FUNCTION_BLOCK FB_OutfeedConveyor
VAR CONSTANT
	sCycleStateTextDef: ARRAY[0..10]  OF STRING :=	
		['State 0: Wait for Start','1','2','3','4','5','6','7','8','9',
		'State 10: Error'];
	
	tCycleStateTimeouts: ARRAY[0..10] OF TIME := 
		[T#10S,T#10S,T#10S,T#10S,T#10S,T#10S,T#10S,T#10S,T#10S,T#10S,
		T#10S];

	sInitStateTextDef: ARRAY[0..10] OF STRING :=
		['State 0: Wait for Start',
		'State 1: Description Init State 1',
		'State 2: Description Init State 2',
		'State 3; Description Init State 3',
		'State 4; Description Init State 4',
		'State 5; Description Init State 5',
		'State 6; Error State'];

	tInitStateTimeouts: ARRAY[0..10] OF TIME := 
		[T#10S,T#10S,T#10S,T#10S,T#10S,T#10S,T#10S,T#10S,T#10S,T#10S
		,T#10S];
END_VAR
VAR_INPUT
	mxResetCycleState				: BOOL;
	mxResetInitState				: BOOL;
	mxForceInit						: BOOL; (*Reset Calibration Flag*)
	mxReset							: BOOL;	(*Reset Error*)
	mxEmergency						: BOOL;
	mxAutoMode						: BOOL; (* TRUE = Automode *)
	mxFirstCycle					: BOOL;

END_VAR
VAR_IN_OUT
	MachParameters					: ST_OutfeedConveyorMachPar;
	ProdParameters					: ST_OutfeedConveyorProdPar;
	SysParameters					: ST_OutfeedConveyorSysPar;
END_VAR
VAR_OUTPUT
	(*Errors*)
	Errors							: ST_OutfeedConveyorErrors;
	mxErrorInit						: BOOL;		(* Error, stop immediately. Initialisation neccesary *)
	mxErrorStopinPos				: BOOL;		(* Error, stop in position. Only reset neccesary *)

(* State vars *)
	mxCycleBusy						: BOOL;
	mxInitBusy						: BOOL;
	
(* Vars *)
	mxInitialized					: BOOL;
	
	mrActModPos						: LREAL;
END_VAR
VAR
(* State vars *)
	miCycleState					: INT :=0;
	miCycleOldstate					: INT :=0;
	mxCycleTransitionState			: BOOL := FALSE;
	sCycleStateText					: STRING;
	exCycleTimeOut					: BOOL;		(* Timeout for the whole programcycle *)
	CycleTimeout					: TON;
	CycleTimeOutUpFlank				: R_TRIG;
	mxCycleTimeoutEnable			: BOOL;
	CycleTime						: REAL;
	mxCycleHasError					: BOOL;
	miStopState						: INT;
	mxStartCycle					: BOOL;
	mxStopCycle						: BOOL;
	mxStopDirect					: BOOL;
	
	miInitState						: INT	:=0;
	miInitOldstate					: INT	:=0;
	mxInitTransitionState			: BOOL	:= FALSE;
	sInitStateText					: STRING;
	exInitTimeOut					: BOOL;		(* Timeout for the whole programcycle *)
	InitTimeout						: TON;
	InitTimeOutUpFlank				: R_TRIG;
	mxInitTimeoutEnable				: BOOL;
	InitTime						: REAL;
	mxInitHasError					: BOOL;
	mxStartInit						: BOOL;
	mxStopInit						: BOOL;
	
	(* Objects *)
	Belt							 : FB_NcAxis;

	mrSetpointPosition				: LREAL;
	mrActPosBeltSaved				: LREAL;
END_VAR

Error();
Cycle();
Init();
Objects();

mrActModPos:= Belt.axAxis.NcToPlc.ModuloActPos;

ACTION Cycle:
(*StateChange (Transition)  Signalgeneration*)
mxCycleTransitionState:=(miCycleState<>miCycleOldstate);
(*State text*)
sCycleStateText:=sCycleStateTextDef[miCycleState];
(*Timeout Watchdog for Statemachine*)
mxCycleTimeoutEnable:=NOT (miCycleState=0) AND NOT mxReset;

CycleTimeout(IN:=mxCycleTimeoutEnable, PT:=tCycleStateTimeouts[miCycleState] );
CycleTimeOutUpFlank(CLK:=CycleTimeout.Q );
miCycleOldstate:=miCycleState;

(*Set Errorbit when Raising edge of Timeout has been detected*)
IF CycleTimeOutUpFlank.Q THEN
	exCycleTimeOut:=TRUE; 			(* 1 Timeout for the whole programcycle *)
END_IF

(*Function to reset the Statemachine*)
IF mxResetCycleState THEN
	mxResetCycleState:= FALSE;
	miCycleState:=0;
	miCycleOldstate:=miCycleState;
	mxCycleTransitionState:=FALSE;

	mxInitialized:= FALSE;
	mxStartCycle:= FALSE;
	mxStopCycle:= FALSE;
	mxStopDirect:= FALSE;
	Belt.M_Stop();
	
END_IF

(*Definition State has Error*)
mxCycleHasError:=FALSE;

(*Cycle State's*)
CASE miCycleState OF
	0:
	(*
		- wait for startcycle
		- Move belt with velo
  
	*)
		IF mxStartCycle THEN
			mxStartCycle:= FALSE;

			miCycleState:= 1;
		END_IF	

	(* Move belt *)
	1:
		IF mxStopDirect THEN
			mxStopDirect:= FALSE;
			
			miCycleState:= 25;
		ELSIF mxStopCycle THEN
			mxStopCycle:= FALSE;

			mrActPosBeltSaved:= Belt.ActPosition;		
	
			miStopState:= miCycleState;
			miCycleState:= 20;
		ELSE
			Belt.M_MoveVelocity(Velocity:= MachParameters.VelocityAuto, Direction:= MC_Positive_Direction);
		END_IF

	(* Stop Cycle, stop belt after x mm*)
	20:
		IF mxStopDirect THEN
			mxStopDirect:= FALSE;
			
			miCycleState:= 25;
		ELSIF Belt.ActPosition > mrActPosBeltSaved + 5000 THEN
			Belt.M_Stop();
			
			miCycleState:= 21;
		ELSE
			Belt.M_MoveVelocity(Velocity:= MachParameters.VelocityAuto, Direction:= MC_Positive_Direction);
		END_IF

	21:
		IF mxStopDirect THEN
			mxStopDirect:= FALSE;
			
			miCycleState:= 25;
		ELSIF NOT Belt.axStatus.Moving OR Belt.axStatus.StandStill THEN
			
			miCycleState:= 0;			
		END_IF

	(* Stop Direct *)
	25:
		mxInitialized:= FALSE;
		mxStartCycle:= FALSE;
		mxStopCycle:= FALSE;
		mxStopDirect:= FALSE;
		
		Belt.M_Stop();

		miCycleState:= 0;
END_CASE

mxCycleBusy:= miCycleState<>0;
END_ACTION

ACTION Error:


(*************************************************************************************************)
mxErrorInit:= FALSE;
mxErrorStopinPos:= Belt.ErrorStop;
END_ACTION

ACTION Init:
(*StateChange (Transition)  Signalgeneration*)
mxInitTransitionState:=(miInitState<>miInitOldstate);
(*State text*)
sInitStateText:=sInitStateTextDef[miInitState];
(*Timeout Watchdog for Statemachine*)
mxInitTimeoutEnable:=NOT (miInitState=0)  AND NOT mxReset;

InitTimeout(IN:=mxInitTimeoutEnable  , PT:=tInitStateTimeouts[miInitState] );
InitTimeOutUpFlank(CLK:=InitTimeout.Q );
miInitOldstate:=miInitState;

(*Set Errorbit when Raising edge of Timeout has been detected*)
IF InitTimeOutUpFlank.Q THEN
	exInitTimeOut:=TRUE; 			(* 1 Timeout for the whole programcycle *)
END_IF

(*Function to reset the Statemachine*)
IF mxResetInitState THEN
	mxResetInitState:=FALSE;
	miInitState:=0;
	miInitOldstate:=miInitState;
	mxInitTransitionState:=FALSE;
	
	mxInitialized:= FALSE;
	mxStartInit:= FALSE;
	mxStopInit:= FALSE;
		
END_IF

(*Definition State has Error*)
mxInitHasError:=FALSE;

(*Init State's*)
CASE miInitState OF
	0:

	(* 
		- Wait for start int
		- Empty belt	
	*)
		IF mxStartInit THEN
			mxStartInit:= FALSE;
			mxInitialized:= FALSE;

			mrSetpointPosition:= Belt.ActPosition + 1000;
			
			miInitState:= 1;
		END_IF

	(* Move, empty belt*)
	1:
		IF mxStopInit THEN
			mxStopInit:= FALSE;
			
			miInitState:= 10;
		ELSIF Belt.M_MoveAbsolute(Position:= mrSetpointPosition, Velocity:= MachParameters.VelocityAuto) THEN
			mxInitialized:= TRUE;

			miInitState:= 0;
		END_IF

	(* Stop Init *)
	10:
		mxInitialized:= FALSE;
		mxStartInit:= FALSE;
		mxStopInit:= FALSE;
		
		Belt.M_Stop();
		
		miInitState:= 0;
			
END_CASE

mxInitBusy:= miInitState<>0;
END_ACTION

METHOD M_StartCycle

IF NOT mxCycleBusy THEN
	mxStartCycle:= TRUE;	
END_IF
END_METHOD

METHOD M_StartInit
VAR_INPUT
END_VAR

IF NOT mxInitBusy THEN
	mxStartInit:= TRUE;
END_IF
END_METHOD

METHOD M_StopCycle

IF mxCycleBusy THEN 
	mxStopCycle:= TRUE; 
END_IF
END_METHOD

METHOD M_StopDirect

IF mxCycleBusy THEN
	mxStopDirect:= TRUE;	
END_IF
END_METHOD

METHOD M_StopInit

IF mxInitBusy THEN 
	mxStopInit:= TRUE; 
END_IF
END_METHOD

ACTION Objects:

Belt(
	mxEnable:= NOT mxEmergency, 
	mxInhibit:= FALSE, 
	mxAutoMode:= mxAutoMode, 
	mxReset:= mxReset, 
	mxEmergency:= mxEmergency, 
	mxSimulation:= , 
	mxFirstCycle:= , 
	mxResetCycle:= , 
	mxDisable_Positive:= FALSE, 
	mxDisable_Negative:= FALSE, 
	mxBlockHMI:= , 
	mrOverride:= 100.0, 
	mrVelocityManual:= MachParameters.VelocityManual, 
	SysParameters:= SysParameters.Belt,
	mxCycleBusy=> , 
	mxRunning=> , 
	Errors=> Errors.NCAxisError, 
	Error=> , 
	ErrorStop=> , 
	axStatus=> , 
	ActPosition=> , 
	ActVelocity=> , 
	axAxis=> );
END_ACTION

END_FUNCTION_BLOCK

(* stored: Version 1.1.0.1, ProductVersion 3.1.4020.12
   POU FB_OutfeedConveyor: Id {b8a7b499-3a0e-47d5-b072-1f1e0bee45c8}, SpecialFunc None
   Action Cycle: Id {b4e2cb85-ce3e-448c-9156-64b284d91ddb}
   Action Error: Id {4b843070-c32e-4e94-909c-b2ec4b0f02b6}
   Action Init: Id {b9fc5455-7ced-4252-a7f2-7e8a2a02f29e}
   Method M_StartCycle: Id {8856c7ab-21a6-495f-9259-f7b3144f553f}
   Method M_StartInit: Id {07e6dfab-bdc1-4744-bb3a-075da4d4af8e}
   Method M_StopCycle: Id {28f51c37-9eb2-466a-9200-d8531abecf71}
   Method M_StopDirect: Id {d998a62d-7ea7-4143-ab81-f1631a5e4166}
   Method M_StopInit: Id {9f266e66-023d-4a2b-8cf2-8dc47cd53205}
   Action Objects: Id {038fd741-a8c6-4fa4-90db-02b38cbe1423} *)
